// Mitsubishi GX Works2 project: Test   PLC: Q06UDH

PROGRAM MAIN
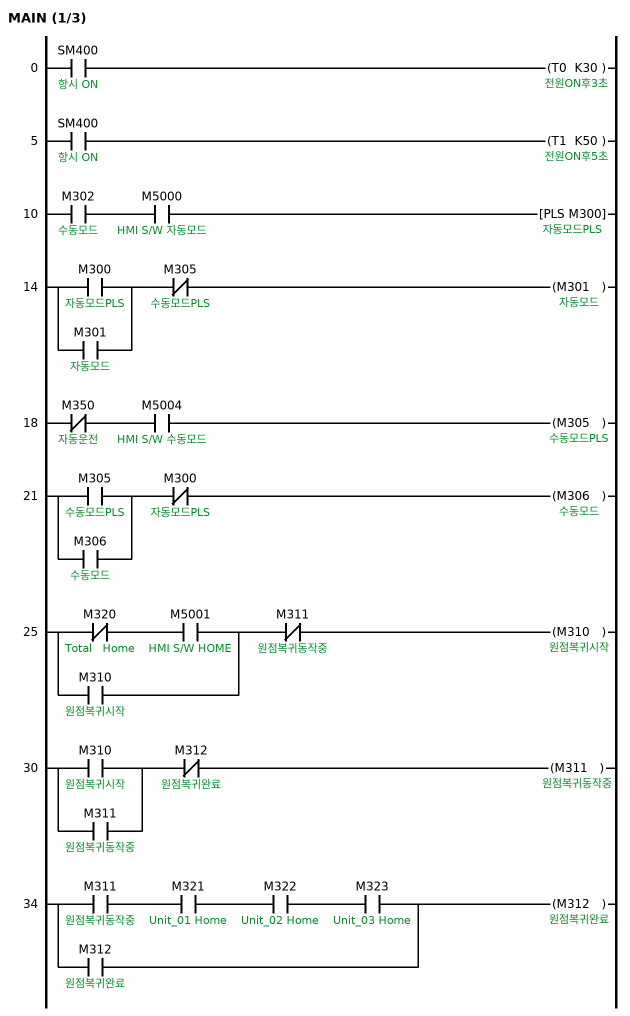
0     LD      SM400  ; 항시 ON
      OUT     T0 K30  ; 전원ON후3초
5     LD      SM400  ; 항시 ON
      OUT     T1 K50  ; 전원ON후5초
10    LD      M302  ; 수동모드
      AND     M5000  ; HMI S/W 자동모드
      PLS     M300  ; 자동모드PLS
14    LD      M300  ; 자동모드PLS
      OR      M301  ; 자동모드
      ANI     M305  ; 수동모드PLS
      OUT     M301  ; 자동모드
18    LDI     M350  ; 자동운전
      AND     M5004  ; HMI S/W 수동모드
      OUT     M305  ; 수동모드PLS
21    LD      M305  ; 수동모드PLS
      OR      M306  ; 수동모드
      ANI     M300  ; 자동모드PLS
      OUT     M306  ; 수동모드
25    LDI     M320  ; Total   Home
      AND     M5001  ; HMI S/W HOME
      OR      M310  ; 원점복귀시작
      ANI     M311  ; 원점복귀동작중
      OUT     M310  ; 원점복귀시작
30    LD      M310  ; 원점복귀시작
      OR      M311  ; 원점복귀동작중
      ANI     M312  ; 원점복귀완료
      OUT     M311  ; 원점복귀동작중
34    LD      M311  ; 원점복귀동작중
      AND     M321  ; Unit_01 Home
      AND     M322  ; Unit_02 Home
      AND     M323  ; Unit_03 Home
      OR      M312  ; 원점복귀완료
      OUT     M312  ; 원점복귀완료
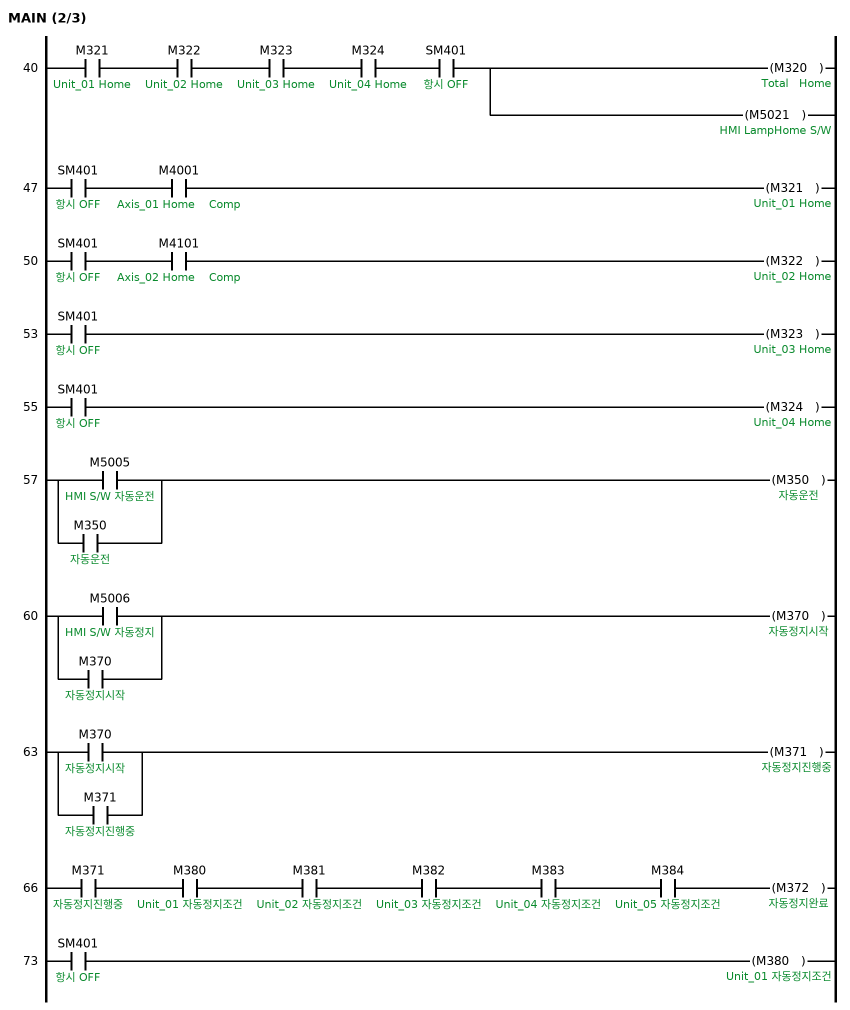
40    LD      M321  ; Unit_01 Home
      AND     M322  ; Unit_02 Home
      AND     M323  ; Unit_03 Home
      AND     M324  ; Unit_04 Home
      AND     SM401  ; 항시 OFF
      OUT     M320  ; Total   Home
      OUT     M5021  ; HMI LampHome S/W
47    LD      SM401  ; 항시 OFF
      AND     M4001  ; Axis_01 Home    Comp
      OUT     M321  ; Unit_01 Home
50    LD      SM401  ; 항시 OFF
      AND     M4101  ; Axis_02 Home    Comp
      OUT     M322  ; Unit_02 Home
53    LD      SM401  ; 항시 OFF
      OUT     M323  ; Unit_03 Home
55    LD      SM401  ; 항시 OFF
      OUT     M324  ; Unit_04 Home
57    LD      M5005  ; HMI S/W 자동운전
      OR      M350  ; 자동운전
      OUT     M350  ; 자동운전
60    LD      M5006  ; HMI S/W 자동정지
      OR      M370  ; 자동정지시작
      OUT     M370  ; 자동정지시작
63    LD      M370  ; 자동정지시작
      OR      M371  ; 자동정지진행중
      OUT     M371  ; 자동정지진행중
66    LD      M371  ; 자동정지진행중
      AND     M380  ; Unit_01 자동정지조건
      AND     M381  ; Unit_02 자동정지조건
      AND     M382  ; Unit_03 자동정지조건
      AND     M383  ; Unit_04 자동정지조건
      AND     M384  ; Unit_05 자동정지조건
      OUT     M372  ; 자동정지완료
73    LD      SM401  ; 항시 OFF
      OUT     M380  ; Unit_01 자동정지조건
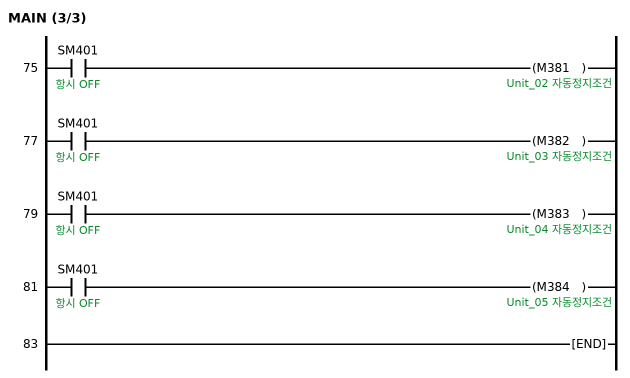
75    LD      SM401  ; 항시 OFF
      OUT     M381  ; Unit_02 자동정지조건
77    LD      SM401  ; 항시 OFF
      OUT     M382  ; Unit_03 자동정지조건
79    LD      SM401  ; 항시 OFF
      OUT     M383  ; Unit_04 자동정지조건
81    LD      SM401  ; 항시 OFF
      OUT     M384  ; Unit_05 자동정지조건
83    END
END_PROGRAM

PROGRAM AutoRun
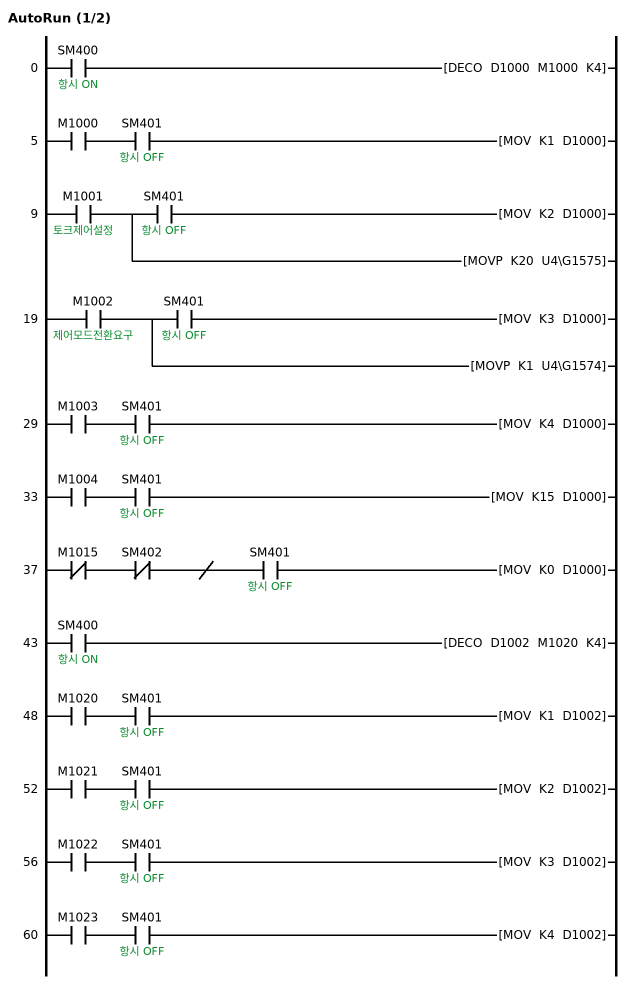
0     LD      SM400  ; 항시 ON
      DECO    D1000 M1000 K4
5     LD      M1000
      AND     SM401  ; 항시 OFF
      MOV     K1 D1000
9     LD      M1001  ; 토크제어설정
      MPS
      AND     SM401  ; 항시 OFF
      MOV     K2 D1000
      MPP
      MOVP    K20 U4\G1575
19    LD      M1002  ; 제어모드전환요구
      MPS
      AND     SM401  ; 항시 OFF
      MOV     K3 D1000
      MPP
      MOVP    K1 U4\G1574
29    LD      M1003
      AND     SM401  ; 항시 OFF
      MOV     K4 D1000
33    LD      M1004
      AND     SM401  ; 항시 OFF
      MOV     K15 D1000
37    LDI     M1015
      ANI     SM402
      INV
      AND     SM401  ; 항시 OFF
      MOV     K0 D1000
43    LD      SM400  ; 항시 ON
      DECO    D1002 M1020 K4
48    LD      M1020
      AND     SM401  ; 항시 OFF
      MOV     K1 D1002
52    LD      M1021
      AND     SM401  ; 항시 OFF
      MOV     K2 D1002
56    LD      M1022
      AND     SM401  ; 항시 OFF
      MOV     K3 D1002
60    LD      M1023
      AND     SM401  ; 항시 OFF
      MOV     K4 D1002
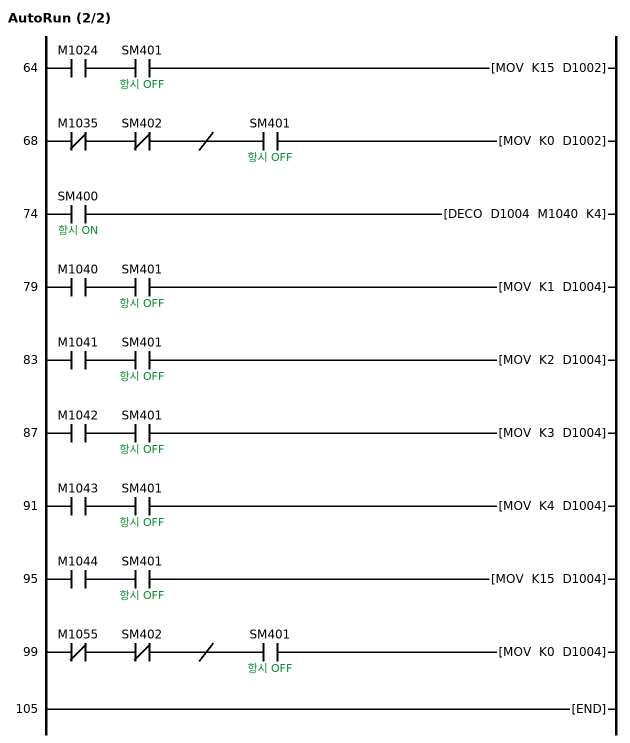
64    LD      M1024
      AND     SM401  ; 항시 OFF
      MOV     K15 D1002
68    LDI     M1035
      ANI     SM402
      INV
      AND     SM401  ; 항시 OFF
      MOV     K0 D1002
74    LD      SM400  ; 항시 ON
      DECO    D1004 M1040 K4
79    LD      M1040
      AND     SM401  ; 항시 OFF
      MOV     K1 D1004
83    LD      M1041
      AND     SM401  ; 항시 OFF
      MOV     K2 D1004
87    LD      M1042
      AND     SM401  ; 항시 OFF
      MOV     K3 D1004
91    LD      M1043
      AND     SM401  ; 항시 OFF
      MOV     K4 D1004
95    LD      M1044
      AND     SM401  ; 항시 OFF
      MOV     K15 D1004
99    LDI     M1055
      ANI     SM402
      INV
      AND     SM401  ; 항시 OFF
      MOV     K0 D1004
105   END
END_PROGRAM

PROGRAM Axis_01
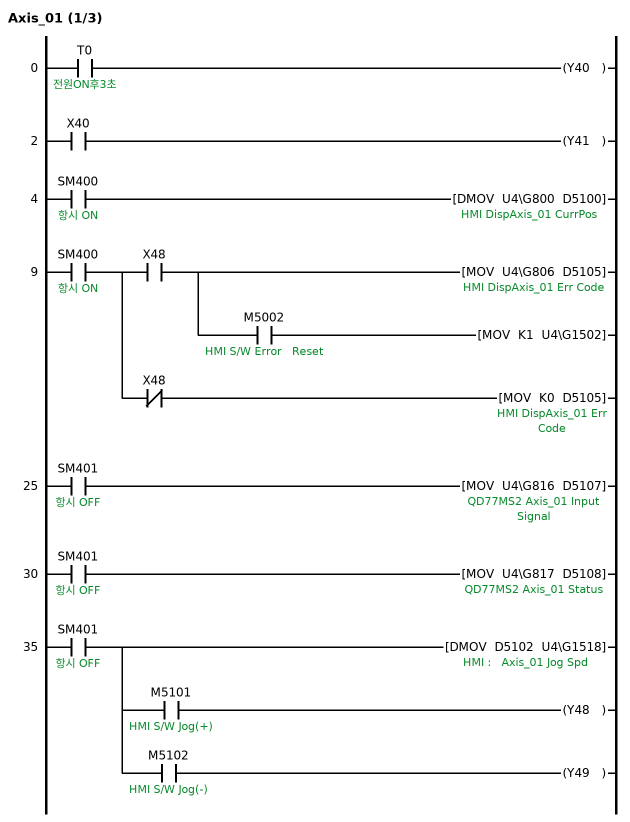
0     LD      T0  ; 전원ON후3초
      OUT     Y40
2     LD      X40
      OUT     Y41
4     LD      SM400  ; 항시 ON
      DMOV    U4\G800 D5100  ; HMI DispAxis_01 CurrPos
9     LD      SM400  ; 항시 ON
      MPS
      AND     X48
      MOV     U4\G806 D5105  ; HMI DispAxis_01 Err Code
      AND     M5002  ; HMI S/W Error   Reset
      MOV     K1 U4\G1502
      MPP
      ANI     X48
      MOV     K0 D5105
25    LD      SM401  ; 항시 OFF
      MOV     U4\G816 D5107  ; QD77MS2 Axis_01 Input   Signal
30    LD      SM401  ; 항시 OFF
      MOV     U4\G817 D5108  ; QD77MS2 Axis_01 Status
35    LD      SM401  ; 항시 OFF
      DMOV    D5102 U4\G1518  ; HMI :   Axis_01 Jog Spd
      MPS
      AND     M5101  ; HMI S/W Jog(+)
      OUT     Y48
      MPP
      AND     M5102  ; HMI S/W Jog(-)
      OUT     Y49
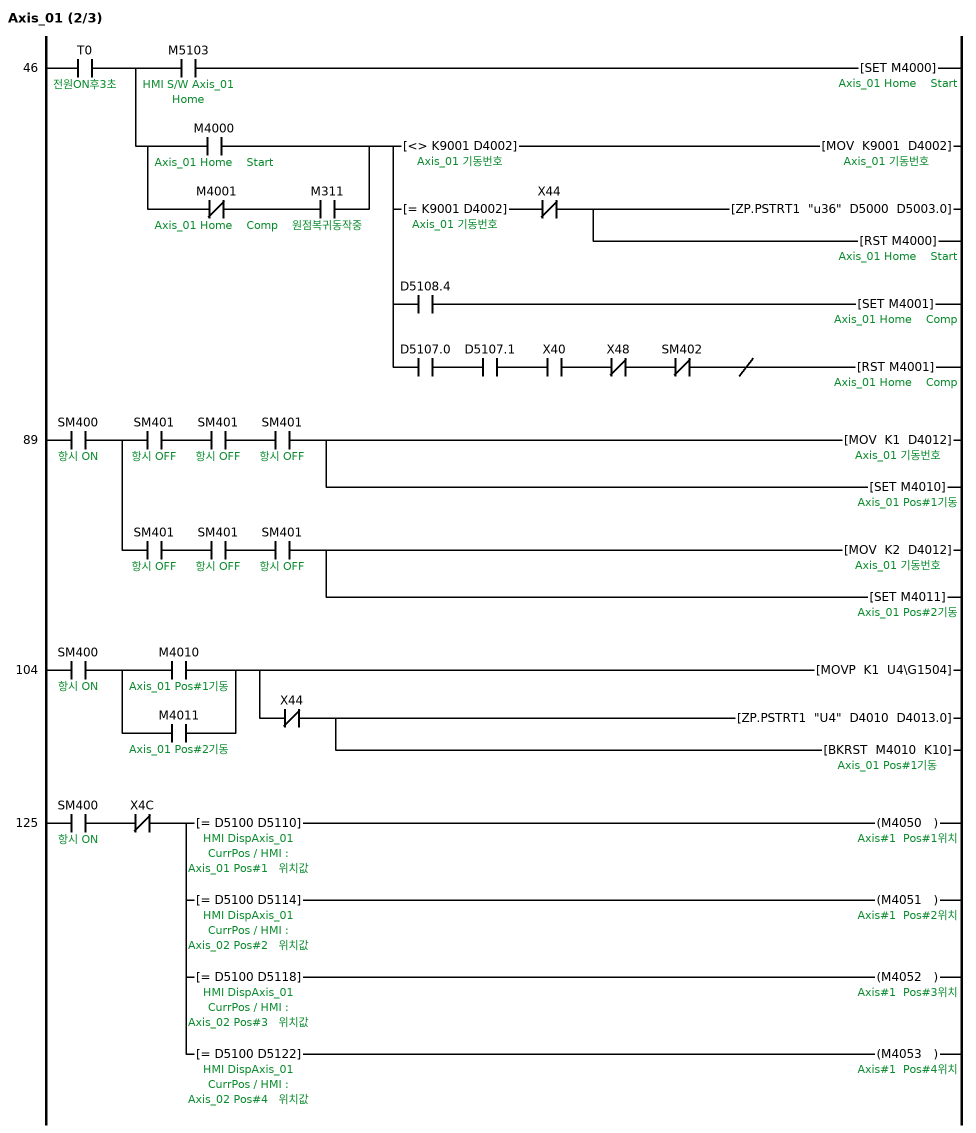
46    LD      T0  ; 전원ON후3초
      MPS
      AND     M5103  ; HMI S/W Axis_01 Home
      SET     M4000  ; Axis_01 Home    Start
      MPP
      LD      M4000  ; Axis_01 Home    Start
      LDI     M4001  ; Axis_01 Home    Comp
      AND     M311  ; 원점복귀동작중
      ORB
      ANB
      MPS
      AND<>   K9001 D4002  ; Axis_01 기동번호
      MOV     K9001 D4002
      MRD
      AND=    K9001 D4002  ; Axis_01 기동번호
      ANI     X44
      ZP.PSTRT1 "u36" D5000 D5003.0
      RST     M4000  ; Axis_01 Home    Start
      MRD
      AND     D5108.4
      SET     M4001  ; Axis_01 Home    Comp
      MPP
      AND     D5107.0
      AND     D5107.1
      AND     X40
      ANI     X48
      ANI     SM402
      INV
      RST     M4001  ; Axis_01 Home    Comp
89    LD      SM400  ; 항시 ON
      MPS
      AND     SM401  ; 항시 OFF
      AND     SM401  ; 항시 OFF
      AND     SM401  ; 항시 OFF
      MOV     K1 D4012  ; Axis_01 기동번호
      SET     M4010  ; Axis_01 Pos#1기동
      MPP
      AND     SM401  ; 항시 OFF
      AND     SM401  ; 항시 OFF
      AND     SM401  ; 항시 OFF
      MOV     K2 D4012
      SET     M4011  ; Axis_01 Pos#2기동
104   LD      SM400  ; 항시 ON
      LD      M4010  ; Axis_01 Pos#1기동
      OR      M4011  ; Axis_01 Pos#2기동
      ANB
      MOVP    K1 U4\G1504
      ANI     X44
      ZP.PSTRT1 "U4" D4010 D4013.0
      BKRST   M4010 K10
125   LD      SM400  ; 항시 ON
      ANI     X4C
      MPS
      AND=    D5100 D5110  ; HMI DispAxis_01 CurrPos / HMI :   Axis_01 Pos#1   위치값
      OUT     M4050  ; Axis#1  Pos#1위치
      MRD
      AND=    D5100 D5114  ; HMI DispAxis_01 CurrPos / HMI :   Axis_02 Pos#2   위치값
      OUT     M4051  ; Axis#1  Pos#2위치
      MRD
      AND=    D5100 D5118  ; HMI DispAxis_01 CurrPos / HMI :   Axis_02 Pos#3   위치값
      OUT     M4052  ; Axis#1  Pos#3위치
      MPP
      AND=    D5100 D5122  ; HMI DispAxis_01 CurrPos / HMI :   Axis_02 Pos#4   위치값
      OUT     M4053  ; Axis#1  Pos#4위치
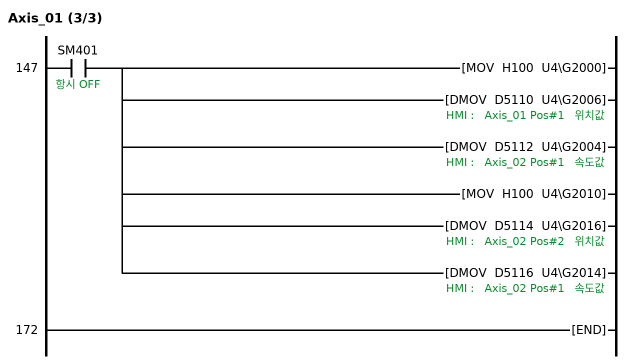
147   LD      SM401  ; 항시 OFF
      MOV     H100 U4\G2000
      DMOV    D5110 U4\G2006
      DMOV    D5112 U4\G2004  ; HMI :   Axis_02 Pos#1   속도값
      MOV     H100 U4\G2010
      DMOV    D5114 U4\G2016
      DMOV    D5116 U4\G2014  ; HMI :   Axis_02 Pos#1   속도값
172   END
END_PROGRAM

PROGRAM Axis_02
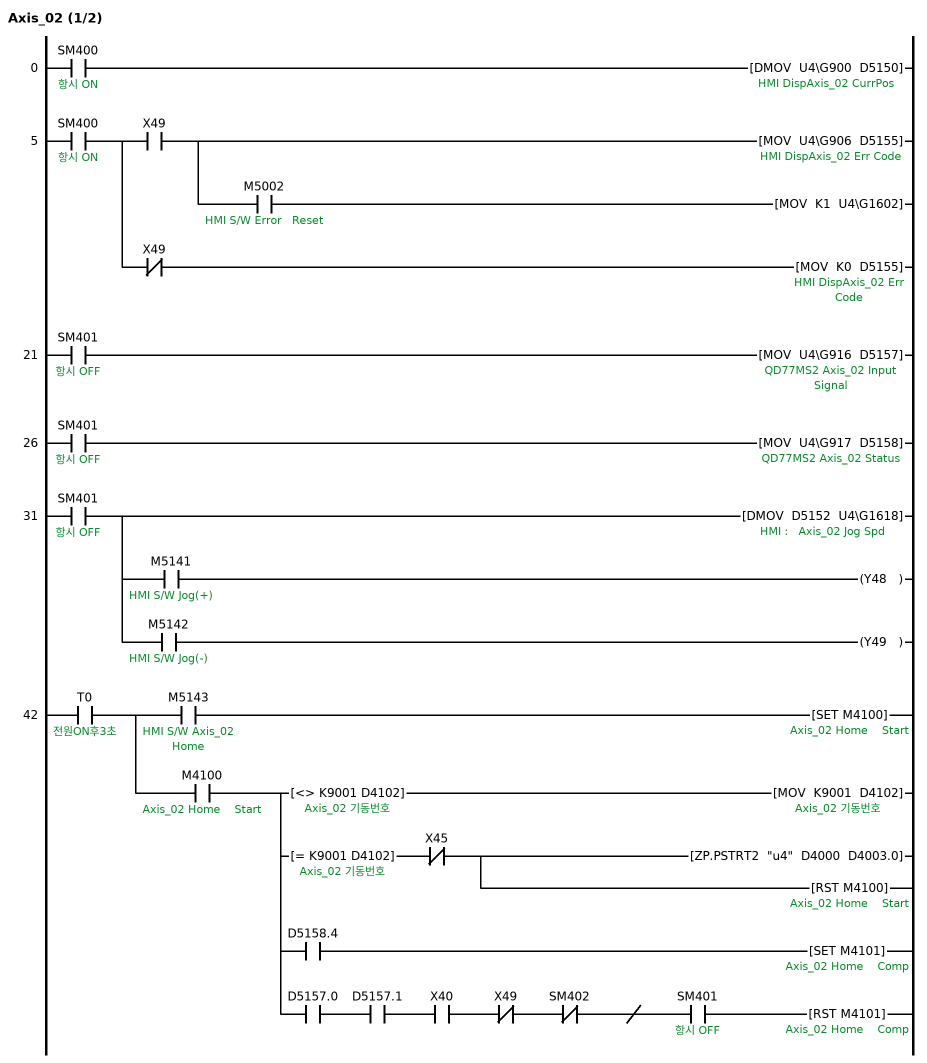
0     LD      SM400  ; 항시 ON
      DMOV    U4\G900 D5150  ; HMI DispAxis_02 CurrPos
5     LD      SM400  ; 항시 ON
      MPS
      AND     X49
      MOV     U4\G906 D5155  ; HMI DispAxis_02 Err Code
      AND     M5002  ; HMI S/W Error   Reset
      MOV     K1 U4\G1602
      MPP
      ANI     X49
      MOV     K0 D5155
21    LD      SM401  ; 항시 OFF
      MOV     U4\G916 D5157  ; QD77MS2 Axis_02 Input   Signal
26    LD      SM401  ; 항시 OFF
      MOV     U4\G917 D5158  ; QD77MS2 Axis_02 Status
31    LD      SM401  ; 항시 OFF
      DMOV    D5152 U4\G1618  ; HMI :   Axis_02 Jog Spd
      MPS
      AND     M5141  ; HMI S/W Jog(+)
      OUT     Y48
      MPP
      AND     M5142  ; HMI S/W Jog(-)
      OUT     Y49
42    LD      T0  ; 전원ON후3초
      MPS
      AND     M5143  ; HMI S/W Axis_02 Home
      SET     M4100  ; Axis_02 Home    Start
      MPP
      AND     M4100  ; Axis_02 Home    Start
      MPS
      AND<>   K9001 D4102  ; Axis_02 기동번호
      MOV     K9001 D4102
      MRD
      AND=    K9001 D4102  ; Axis_02 기동번호
      ANI     X45
      ZP.PSTRT2 "u4" D4000 D4003.0
      RST     M4100  ; Axis_02 Home    Start
      MRD
      AND     D5158.4
      SET     M4101  ; Axis_02 Home    Comp
      MPP
      AND     D5157.0
      AND     D5157.1
      AND     X40
      ANI     X49
      ANI     SM402
      INV
      AND     SM401  ; 항시 OFF
      RST     M4101  ; Axis_02 Home    Comp
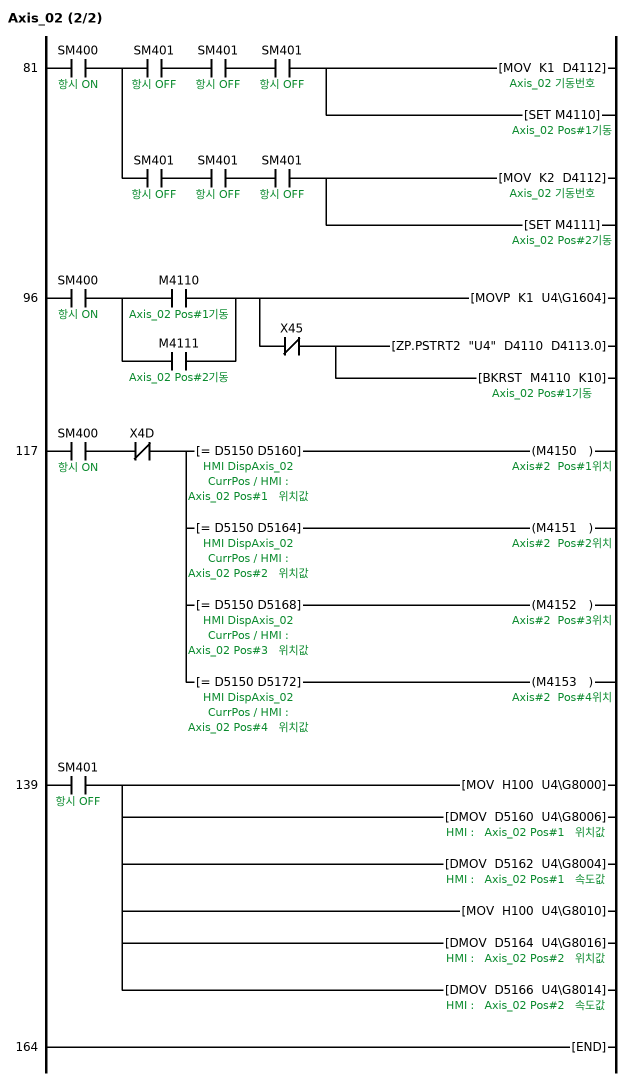
81    LD      SM400  ; 항시 ON
      MPS
      AND     SM401  ; 항시 OFF
      AND     SM401  ; 항시 OFF
      AND     SM401  ; 항시 OFF
      MOV     K1 D4112  ; Axis_02 기동번호
      SET     M4110  ; Axis_02 Pos#1기동
      MPP
      AND     SM401  ; 항시 OFF
      AND     SM401  ; 항시 OFF
      AND     SM401  ; 항시 OFF
      MOV     K2 D4112
      SET     M4111  ; Axis_02 Pos#2기동
96    LD      SM400  ; 항시 ON
      LD      M4110  ; Axis_02 Pos#1기동
      OR      M4111  ; Axis_02 Pos#2기동
      ANB
      MOVP    K1 U4\G1604
      ANI     X45
      ZP.PSTRT2 "U4" D4110 D4113.0
      BKRST   M4110 K10
117   LD      SM400  ; 항시 ON
      ANI     X4D
      MPS
      AND=    D5150 D5160  ; HMI DispAxis_02 CurrPos / HMI :   Axis_02 Pos#1   위치값
      OUT     M4150  ; Axis#2  Pos#1위치
      MRD
      AND=    D5150 D5164  ; HMI DispAxis_02 CurrPos / HMI :   Axis_02 Pos#2   위치값
      OUT     M4151  ; Axis#2  Pos#2위치
      MRD
      AND=    D5150 D5168  ; HMI DispAxis_02 CurrPos / HMI :   Axis_02 Pos#3   위치값
      OUT     M4152  ; Axis#2  Pos#3위치
      MPP
      AND=    D5150 D5172  ; HMI DispAxis_02 CurrPos / HMI :   Axis_02 Pos#4   위치값
      OUT     M4153  ; Axis#2  Pos#4위치
139   LD      SM401  ; 항시 OFF
      MOV     H100 U4\G8000
      DMOV    D5160 U4\G8006
      DMOV    D5162 U4\G8004  ; HMI :   Axis_02 Pos#1   속도값
      MOV     H100 U4\G8010
      DMOV    D5164 U4\G8016
      DMOV    D5166 U4\G8014  ; HMI :   Axis_02 Pos#2   속도값
164   END
END_PROGRAM

PROGRAM Error
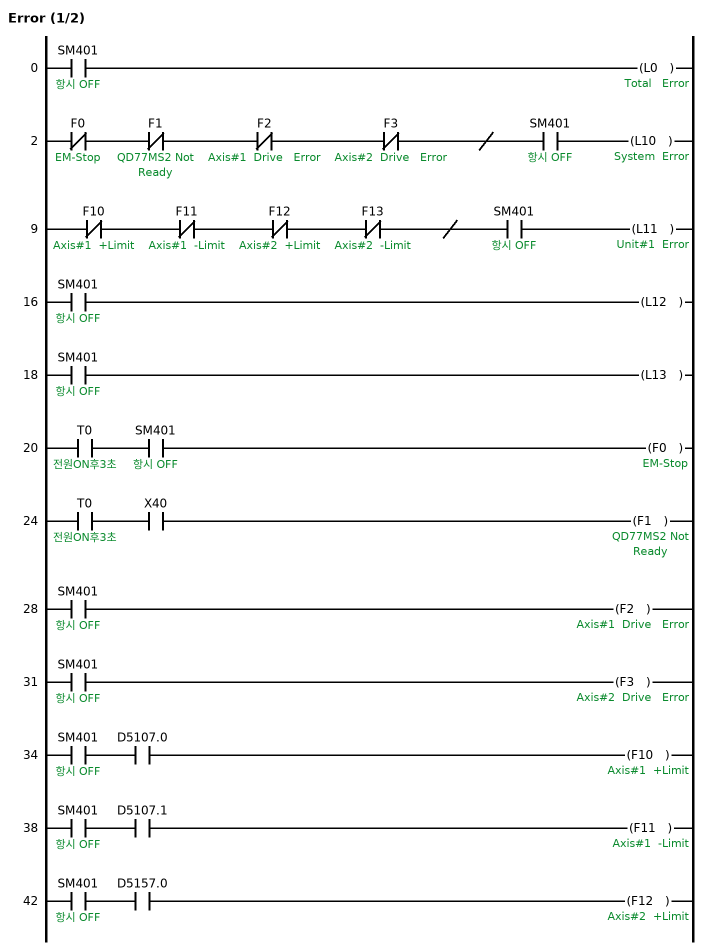
0     LD      SM401  ; 항시 OFF
      OUT     L0  ; Total   Error
2     LDI     F0  ; EM-Stop
      ANI     F1  ; QD77MS2 Not     Ready
      ANI     F2  ; Axis#1  Drive   Error
      ANI     F3  ; Axis#2  Drive   Error
      INV
      AND     SM401  ; 항시 OFF
      OUT     L10  ; System  Error
9     LDI     F10  ; Axis#1  +Limit
      ANI     F11  ; Axis#1  -Limit
      ANI     F12  ; Axis#2  +Limit
      ANI     F13  ; Axis#2  -Limit
      INV
      AND     SM401  ; 항시 OFF
      OUT     L11  ; Unit#1  Error
16    LD      SM401  ; 항시 OFF
      OUT     L12
18    LD      SM401  ; 항시 OFF
      OUT     L13
20    LD      T0  ; 전원ON후3초
      AND     SM401  ; 항시 OFF
      OUT     F0  ; EM-Stop
24    LD      T0  ; 전원ON후3초
      AND     X40
      OUT     F1  ; QD77MS2 Not     Ready
28    LD      SM401  ; 항시 OFF
      OUT     F2  ; Axis#1  Drive   Error
31    LD      SM401  ; 항시 OFF
      OUT     F3  ; Axis#2  Drive   Error
34    LD      SM401  ; 항시 OFF
      AND     D5107.0
      OUT     F10  ; Axis#1  +Limit
38    LD      SM401  ; 항시 OFF
      AND     D5107.1
      OUT     F11  ; Axis#1  -Limit
42    LD      SM401  ; 항시 OFF
      AND     D5157.0
      OUT     F12  ; Axis#2  +Limit
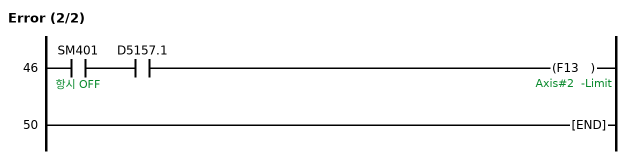
46    LD      SM401  ; 항시 OFF
      AND     D5157.1
      OUT     F13  ; Axis#2  -Limit
50    END
END_PROGRAM
